// Mitsubishi GX Works2 project: DIMACULANGAN_PLC_finals   PLC: FX1N/FX1NC

PROGRAM MAIN
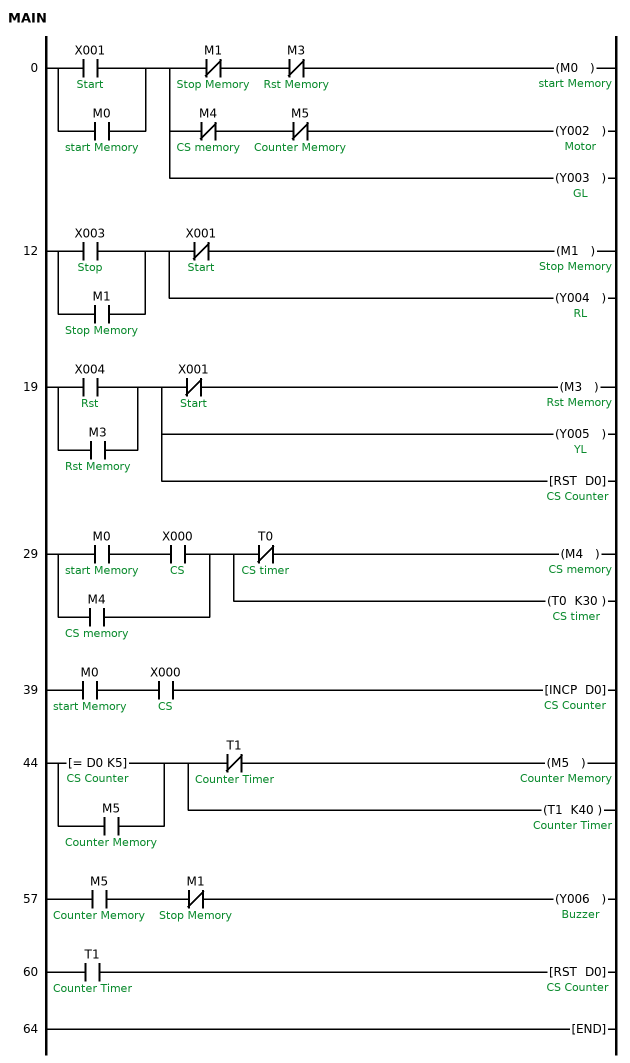
0     LD      X001  ; Start
      OR      M0  ; start Memory
      MPS
      ANI     M1  ; Stop Memory
      ANI     M3  ; Rst Memory
      OUT     M0  ; start Memory
      MRD
      ANI     M4  ; CS memory
      ANI     M5  ; Counter Memory
      OUT     Y002  ; Motor
      MPP
      OUT     Y003  ; GL
12    LD      X003  ; Stop
      OR      M1  ; Stop Memory
      MPS
      ANI     X001  ; Start
      OUT     M1  ; Stop Memory
      MPP
      OUT     Y004  ; RL
19    LD      X004  ; Rst
      OR      M3  ; Rst Memory
      MPS
      ANI     X001  ; Start
      OUT     M3  ; Rst Memory
      MPP
      OUT     Y005  ; YL
      RST     D0  ; CS Counter
29    LD      M0  ; start Memory
      AND     X000  ; CS
      OR      M4  ; CS memory
      MPS
      ANI     T0  ; CS timer
      OUT     M4  ; CS memory
      MPP
      OUT     T0 K30  ; CS timer
39    LD      M0  ; start Memory
      AND     X000  ; CS
      INCP    D0
44    LD=     D0 K5  ; CS Counter
      OR      M5  ; Counter Memory
      MPS
      ANI     T1  ; Counter Timer
      OUT     M5  ; Counter Memory
      MPP
      OUT     T1 K40  ; Counter Timer
57    LD      M5  ; Counter Memory
      ANI     M1  ; Stop Memory
      OUT     Y006  ; Buzzer
60    LD      T1  ; Counter Timer
      RST     D0  ; CS Counter
64    END
END_PROGRAM
